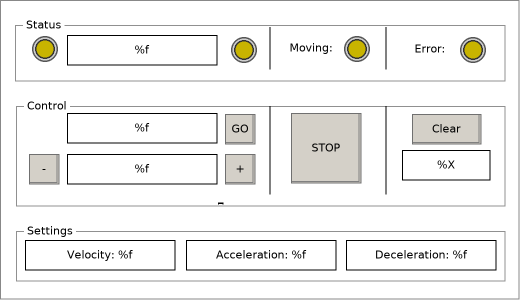
VISUALIZATION VISU_MotionStage  // 520x300
VAR_IN_OUT
	VisuMotionStage: DUT_MotionStage;
	Extras: DUT_MotionStage_Extras;
END_VAR
    GroupBox (15,17 490x64), "Status"
        Lamp1 (15,17 30x30), tooltip "Low Limit Hit Indicator", variable: Extras.bVisuLowLim, style: Lamp-Lamp1-Yellow
        Rectangle (52,18 150x30), "%f", tooltip "Current Position", text variable: VisuMotionStage.stAxisStatus.fActPosition
        Lamp1 (214,18 30x30), tooltip "High Limit Hit Indicator", variable: Extras.bVisuHighLim, style: Lamp-Lamp1-Yellow
        Lamp1 (327,17 30x30), variable: VisuMotionStage.bBusy, style: Lamp-Lamp1-Yellow
        Label (262,16 68x30), "Moving:"
        Line (371,52) (371,10)
        Lamp1 (443,18 30x30), variable: VisuMotionStage.bError, style: Lamp-Lamp1-Yellow
    Rectangle (218,203 5x0)
    GroupBox (16,98 489x108), "Control"
        Rectangle (51,15 150x30), "%f", tooltip "Set Position", text variable: VisuMotionStage.fPosition
            OnMouseDown: write the text variable via Default
        Button (13,56 30x30), "-"
            OnMouseDown: execute {
                VisuMotionStage.nCommand := 3;
                VisuMotionStage.fPosition := VisuMotionStage.stAxisStatus.fActPosition - Extras.fVisuStep;
                VisuMotionStage.bExecute := TRUE;
            }
        Rectangle (51,56 150x30), "%f", tooltip "Step Size", text variable: Extras.fVisuStep
            OnMouseDown: write the text variable via Default
        Button (209,16 30x30), "GO", tooltip "GO to set position"
            OnMouseDown: execute { VisuMotionStage.nCommand := 3; VisuMotionStage.bExecute := TRUE; }
        Line (254,96) (254,8)
        Line (370,96) (370,8)
        Button (396,16 69x30), "Clear"
            tap VisuMotionStage.bReset
        Button (275,15 70x70), "STOP", tooltip "GO to set position"
            OnMouseDown: execute { VisuMotionStage.bExecute := FALSE; }
        Button (209,56 30x30), "+"
            OnMouseDown: execute {
                VisuMotionStage.nCommand := 3;
                VisuMotionStage.fPosition := VisuMotionStage.stAxisStatus.fActPosition + Extras.fVisuStep;
                VisuMotionStage.bExecute := TRUE;
            }
    GroupBox (16,223 489x58), "Settings"
        Rectangle (9,17 150x30), "Velocity: %f", text variable: VisuMotionStage.fVelocity
            OnMouseDown: write the text variable via Default
        Rectangle (170,17 150x30), "Acceleration: %f", tooltip "0 = Default Acceleration", text variable: VisuMotionStage.fAcceleration
            OnMouseDown: write the text variable via Default
        Rectangle (330,17 150x30), "Deceleration: %f", tooltip "0 = Default Deceleration", text variable: VisuMotionStage.fDeceleration
            OnMouseDown: write the text variable via Default
    Line (270,69) (270,27)
    Label (396,34 68x30), "Error:"
    Rectangle (402,150 88x30), "%X", tooltip "Error Code", text variable: VisuMotionStage.stAxisStatus.nErrorId
END_VISUALIZATION

(* stored: Version 1.1.0.1, ProductVersion 3.1.4022.12
   Visu VISU_MotionStage: Id {f7de9cfd-6d88-430a-8070-305db7bc83b0} *)
